{attribute 'GeneratedUsingTerminal: EJ5002-0000-0017'}
{attribute addProperty BoxType "EJ5002-0000-0017"}
{attribute addProperty Id "SSI_Inputs_Channel_1AT %I*SSI_Inputs_Channel_EDA1628411SSI_Inputs_Channel_2AT %I*SSI_Inputs_Channel_EDA1628411WcStateAT %I*WcState_9091E0EB2InfoDataAT %I*InfoData_94A18F5E2"}
{attribute addProperty CRC "1007138389"}
{attribute addProperty Size "26"}
TYPE EJ5002_3C07B655 EXTENDS EtcSlaveTerminalBase_947E5A46 :
STRUCT
	{attribute addProperty Name "SSI_Inputs_Channel_1"}
	SSI_Inputs_Channel_1 : SSI_Inputs_Channel_EDA16284;
	{attribute addProperty Name "SSI_Inputs_Channel_2"}
	SSI_Inputs_Channel_2 : SSI_Inputs_Channel_EDA16284;
	{attribute addProperty Name "WcState"}
	WcState : WcState_9091E0EB;
	{attribute addProperty Name "InfoData"}
	InfoData : InfoData_94A18F5E;
END_STRUCT
END_TYPE

(* stored: Version 1.2.0.0, ProductVersion 3.1.4024.9
   DUT EJ5002_3C07B655: Id {cf87d464-435a-4a1a-a39c-9d087b654c13} *)
